(* Logix 5000 project; controller CancelaAutomotivaParte1 vendor 1 type 14 code 89 rev 20.12; software revision 20.05 *)

TASK MainTask (continuous, watchdog 500 ms) : MainProgram

MODULES
   Controller : vendor 1 type 14 code 89 (CompactLogixL23E_QBFC1_Controller 0, rev 20.12)
      LocalENB : vendor 1 type 12 code 191 (CompactLogixL23E_QBFC1_Ethernet 1, rev 20.11)
      Local : CompactBus (CompactVirtualAdapter 3, rev 20.11)
         Discrete_Inputs : vendor 1 type 7 code 320 (Compact 1, rev 3.1, Input RPI 20 ms)
         Discrete_Outputs : vendor 1 type 7 code 322 (Compact 2, rev 3.1, Output RPI 20 ms)
         Analog_IO : vendor 1 type 10 code 120 (Compact 3, rev 1.1, Output RPI 80 ms)
         Counters : vendor 1 type 109 code 70 (Compact 4, rev 1.1, Output RPI 20 ms)
END_MODULES

PROGRAM MainProgram   (* main routine MainRoutine *)
VAR
   AbrirCancela : ALIAS FOR Local:2:O.Data.1;
   AcessoPermitido : BOOL;
   BDPresencaCarro : BOOL;
   CancelaAberta : BOOL;
   CarroPassando : BOOL;
   CarroPassou : BOOL;
   FecharCancela : ALIAS FOR Local:2:O.Data.2;
   LeituraCracha : ALIAS FOR Local:1:I.Data.1;
   PresencaCarro : ALIAS FOR Local:1:I.Data.4;
   StartStop : ALIAS FOR Local:1:I.Data.3;
   TempoDescida : TIMER := (PRE := 5000);
   TempoEspera : TIMER := (PRE := 10000);
   TempoSubida : TIMER := (PRE := 5000);
END_VAR

ROUTINE MainRoutine   (* ladder *)
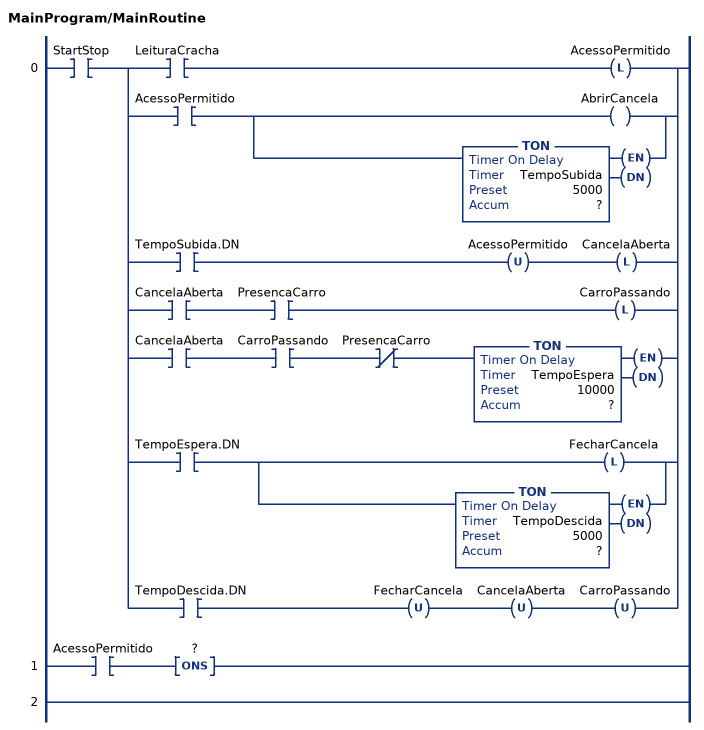
   0: XIC(StartStop)[[[[[XIC(LeituraCracha) OTL(AcessoPermitido) ,XIC(AcessoPermitido) [OTE(AbrirCancela) ,TON(TempoSubida,?,?) ] ] ,XIC(TempoSubida.DN) OTU(AcessoPermitido) OTL(CancelaAberta) ] ,XIC(CancelaAberta) XIC(PresencaCarro) OTL(CarroPassando) ] ,XIC(CancelaAberta) XIC(CarroPassando) XIO(PresencaCarro) TON(TempoEspera,?,?) ] ,[XIC(TempoEspera.DN) [OTL(FecharCancela) ,TON(TempoDescida,?,?) ] ,XIC(TempoDescida.DN) OTU(FecharCancela) OTU(CancelaAberta) OTU(CarroPassando) ] ];
   1: XIC(AcessoPermitido)ONS(?);
   2: ;
END_ROUTINE
END_PROGRAM
